// TIA Portal V17 export
// export: Created 2025-03-10T12:16:40.9467039Z, ExportSetting WithDefaults, DisplayName Totally Integrated Automation Portal, DisplayVersion V17 Update 8, DisplayName TIA Portal Openness, DisplayVersion V17 Update 8, DisplayName TIA Portal Version Control Interface, DisplayVersion V17, DisplayName SINAMICS Startdrive Advanced, DisplayVersion V17 SP2, DisplayName SINAMICS Startdrive G110M, G120, G120C, G120D, G120P, G115D, DisplayVersion V17 SP2, DisplayName SINAMICS Startdrive G130, G150, S120, S150, SINAMICS MV, S210, DisplayVersion V17 SP2, DisplayName STEP 7 Professional, DisplayVersion V17 Update 8, DisplayName SINUMERIK ONE STEP 7 Toolbox, DisplayVersion V17 Update 12, DisplayName SINUMERIK 840D sl STEP 7 Toolbox, DisplayVersion V17 Update 12, DisplayName STEP 7 Safety, DisplayVersion V17 Update 6, DisplayName WinCC Advanced, DisplayVersion V17 Update 8
DATA_BLOCK "LTLP_SLModuleDiagnosticDB"   // DB595
{ DB_Accessible_From_OPC_UA := 'FALSE' }
// stored: AutoNumber true, DBAccessibleFromOPCUA false, DBAccessibleFromWebserver true, InstanceOfName LTLP_SLModuleDiagnostic, InstanceOfType FB
"LTLP_SLModuleDiagnostic"
   // VAR_INPUT
   //    DeviceAdress : HW_ANY;
   //    ReadData : Bool;
   //    RestartPLC : Bool;
   // END_VAR
   // VAR_OUTPUT
   //    IsBusy : Bool;
   //    Done : Bool;
   //    RET_VALUE : Word;
   // END_VAR
   // VAR
   //    stNewDataSaved : UInt;
   //    stCountOfDevicesFound : Int;
   //    stCountOfConfiguredModuls : Int;
   //    stCountOfFailedModuls : Int;
   //    stCountOfDisabledModuls : Int;
   //    stCountOfExistingModuls : Int;
   //    stCountOfModulsWithProblems : Int;
   //    stDiagnosticCPU { S7_SetPoint := 'True'} : Array[0..31] of "LTLP_typeSLModuleDiagnostic";
   //    stInstGetNameOfDevice { S7_SetPoint := 'True'} : Get_Name;
   //    stInstGeoAddressIOSystem { S7_SetPoint := 'True'} : GEOADDR;
   //    stDiagnosticDataMode { S7_SetPoint := 'True'} : DWord;
   //    stDiagnosticDataDevice : DIS;
   //    stDiagnosticDataModule { S7_SetPoint := 'True'} : DNN;
   //    stDevicesChecked { S7_SetPoint := 'True'} : Bool;
   //    stCheckCPUData : Bool;
   //    stCheckNextDevice : Int;
   //    stCheckDeviceFound : Int;
   //    stImpStartNewRead { S7_SetPoint := 'True'} : Bool;
   //    stTrigStartNewRead : Bool;
   //    stReadDataSaved : Bool;
   //    stGetDiagLADDR : HW_ANY;
   //    stGetDiagCNT_DIAG : UInt;
   //    stGetDiagRetvalue : Int;
   //    stLog2GeoRetValue : Int;
   //    stReadDataChanged { S7_SetPoint := 'True'} : Int;
   // END_VAR
BEGIN
END_DATA_BLOCK
